FUNCTION FC_Check_EOT : BOOL
VAR_INPUT
	I_sString : REFERENCE TO T_MaxString;
END_VAR
VAR
	stringPos	: INT;
END_VAR

stringPos := FIND(I_sString, EOT);
IF stringPos <> 0 THEN
	I_sString := MID(I_sString, stringPos-1, 1);
	FC_Check_EOT := TRUE;
ELSE
	FC_Check_EOT := FALSE;
END_IF

END_FUNCTION

(* stored: Version 1.1.0.1, ProductVersion 3.1.4024.15
   POU FC_Check_EOT: Id {13103aff-fdcf-4310-bc8e-5635153fad3d}, SpecialFunc None *)
